FUNCTION_BLOCK FB_OptimizePID

VAR_INPUT
	// Starts the sequence on the rising edge
	Enable : BOOL; 
	// Set point 
	ProcessSetpoint : REAL; 
	// Process measurement 
	ProcessValue : REAL;
	// Number of automatic adjustment cycles (minimum 2) 
	NumCycles : INT := 2; 
	// Reset
	Reset : BOOL;
	// Low value for the square wave output
	ControlLowVal : REAL;
	// High value for the square wave output
	ControlHighVal: REAL;
	// PID constants to use
	PIDType: E_PIDOptimizationType;
END_VAR
VAR_OUTPUT
	// End sequence
	TuningDone: BOOL;
	// Square wave output for the exitation of the process
	ControlValue: REAL; 
	// Proportional gain
	Kp: REAL;
	// Integral time in S
	Ki: REAL;
	// Derivative time in s
	Kd: REAL;
	// Ultimate Gain 
	Ku: REAL;
	// Ultimate Period
	Tu: REAL;
END_VAR
VAR
	// Enable trigger
	rTrigEnable : R_TRIG;
	// Amplitude of process variable
	b: REAL;
	// Amplitude of control variable
	a: REAL;
    TuFreq: FB_FreqMeasure;      
    b_Min: REAL;
    b_Max: REAL;
	EndTrigger : R_TRIG;    
    TuningSequence: E_PIDOptimizationStage;
    CycleNumber: INT;
END_VAR
VAR CONSTANT
    PI : REAL := REAL#3.14159265358979323846264338327950288;
	REAL_MAX : REAL :=  3.402823E+38;
	REAL_MIN : REAL :=-3.402823E+38;
END_VAR


IF Reset THEN
    TuningSequence := E_PIDOptimizationStage.Init;
	TuningDone := FALSE;
END_IF;
IF TuningDone THEN
	RETURN;
END_IF

CASE TuningSequence OF
	// Startup - initialize and set to ramp up to setpoint
	E_PIDOptimizationStage.Init: 
		ControlValue := ControlLowVal;
		IF rTrigEnable.Q THEN
			TuFreq(
				IN := FALSE,
				PERIODS := NumCycles,
				RESET := TRUE); 
			b_Min := REAL_MAX ;
			b_Max := REAL_MIN ;
			KP := 0;
			Ki := 0;
			Kd := 0;
			CycleNumber := 0;
			TuningSequence := E_PIDOptimizationStage.RampingUp;
		END_IF;

	// Ramp to setpoint
	E_PIDOptimizationStage.RampingUp:
		ControlValue := ControlHighVal;
		// If we hit the setpoint, transition to ramping down
		IF ProcessValue > ProcessSetpoint THEN
			ControlValue := ControlLowVal;
			CycleNumber := CycleNumber + 1;
			TuningSequence := E_PIDOptimizationStage.RampingDown;
		END_IF;
		
	// Wait for process value to fall below setpoint
	E_PIDOptimizationStage.RampingDown:
		// Once process value falls, either we are done if we hit the cycle count,
		// or we need to start the next cycle.
		IF ProcessValue < ProcessSetpoint THEN
			IF CycleNumber > NumCycles THEN
				TuningSequence := E_PIDOptimizationStage.Done;
			ELSE
				TuningSequence := E_PIDOptimizationStage.RampingUp;
			END_IF;
		END_IF;

END_CASE;


(*Only Start Measuring Min/Max once we've crossed setpoint once this is to make sure we don't take 0 as value*)
IF CycleNumber  > 0  THEN
	b_Min := MIN(b_Min, ProcessValue);
	b_Max := MAX(b_Max, ProcessValue);
	
	
	TuFreq(
		IN := ProcessValue > ProcessSetpoint,
		PERIODS := NumCycles,
		RESET := FALSE); 
	// We don't check the error becuase i'm lazy. In a real system, if the TuFreq goes invalid, it means the data is screwed up and you need to do something.

END_IF
EndTrigger(CLK := TuningSequence = E_PIDOptimizationStage.Done AND TuFreq.OUT <> 0);
IF EndTrigger.Q THEN
    // Calculate amplitude of control variable
    a := ControlHighVal - ControlLowVal;

	// Calculate amplitude of process variable
    b := b_Max - b_Min;

    // Calculate ultimate period and gain
    Ku := (4 * b)/(PI * a);
    Tu := 1 / TuFreq.OUT;

    CASE PIDType OF
    E_PIDOptimizationType.PessenIntegralRule:
        Kp := 0.7 * Ku;
        Ki := (1.75 * Kp) / Tu;
        Kd := 3* Kp * (Tu/20.0);

    E_PIDOptimizationType.SomeOvershoot:
        Kp := Ku /3.0;
        Ki := (2/3.0) * Ku / Tu ;
        Kd := Ku * Tu  / 10.0;

    E_PIDOptimizationType.NoOvershoot:
        Kp := 0.2 * Ku ;
        Ki := 2 * Ku / Tu  / 5.0;
        Kd := 2* Ku * Tu / 3.0;
    END_CASE;
    
    TuningDone := TRUE;
    TuningSequence := E_PIDOptimizationStage.Init;

END_IF;
rTrigEnable(CLK := Enable);

END_FUNCTION_BLOCK

(* stored: Version 1.1.0.1, ProductVersion 3.1.4022.16
   POU FB_OptimizePID: Id {626227d0-9b37-4afe-a71a-fd287754eb95}, SpecialFunc None *)
